//{{V2}}
ORGANIZATION_BLOCK OB1
TITLE= "Zyklisches Hauptprogramm"
//Längenerkennung durch 2 Lichtschranken
//
//Kurz:
//____
//____
//
//
//Lang:
//   __
//__|  |__
//   __
//__|  |__


AUTHOR:nb
FAMILY:nb
NAME:nb
VERSION:1.0


VAR_TEMP
       OB1_EV_CLASS:BYTE //Bits 0-3 = 1 (Coming event), Bits 4-7 = 1 (Event class 1)
       OB1_SCAN_1:BYTE //1 (Cold restart scan 1 of OB 1), 3 (Scan 2-n of OB 1)
       OB1_PRIORITY:BYTE //1 (Priority of 1 is lowest)
       OB1_OB_NUMBR:BYTE //1 (Organization block 1, OB1)
       OB1_RESERVED_1:BYTE //Reserved for system
       OB1_RESERVED_2:BYTE //Reserved for system
       OB1_PREV_CYCLE:INT //Cycle time of previous OB1 scan (milliseconds)
       OB1_MIN_CYCLE:INT //Minimum cycle time of OB1 (milliseconds)
       OB1_MAX_CYCLE:INT //Maximum cycle time of OB1 (milliseconds)
       OB1_DATE_TIME:DATE_AND_TIME //Date and time OB1 started
END_VAR
BEGIN

NETWORK
TITLE=Kurze Kiste setzen
//{{k}}

       UN   E       124.1
       U(
       U    E       124.2
       FP   M        20.0
       )
       S    A       125.0
NETWORK
TITLE=Kurze Kiste zurücksetzen
//{{k}}

       O    A124.0
       ON   E       124.0
       FP   M        20.5
       R    A       125.0
NETWORK
TITLE=Lange Kiste setzen
//{{k}}

       U    E124.1
       U(
       U    E124.2
       FP   M        20.1
       )
       S    A124.0
NETWORK
TITLE=Lange Kiste rücksetzen
//{{k}}

       O    A125.0
       ON   E124.0
       FP   M        20.4
       R    A124.0
END_ORGANIZATION_BLOCK
